{attribute 'GeneratedUsingTerminal: EL3773-0000-0016'}
{attribute addProperty BoxType "EL3773-0000-0016"}
{attribute addProperty Id "I2_SAMPLESAT %I*I2_SAMPLES_2D13B74B20"}
{attribute addProperty CRC "109000063"}
{attribute addProperty Size "20"}
TYPE L2_Current_Samples_067F357F EXTENDS InputBase_8311D824 :
STRUCT
	{attribute addProperty Name "I2_SAMPLES"}
	I2_SAMPLES AT %I* : I2_SAMPLES_2D13B74B;
END_STRUCT
END_TYPE

(* stored: Version 1.2.0.0, ProductVersion 3.1.4024.9
   DUT L2_Current_Samples_067F357F: Id {ab4f74cc-c9fe-4ffa-80a5-5e7bbaaee32a} *)
